{attribute 'qualified_only'}
VAR_GLOBAL
	dOut AT%Q* :ARRAY[1..16]OF BOOL;
	dIn  AT%I* :ARRAY[1..24]OF BOOL;
END_VAR

(* stored: Version 1.1.0.1, ProductVersion 3.1.4026.18
   GVL GVL_IO: Id {b17cdcaf-0338-4dc3-b0f8-36248c1bde3a} *)
